Omron CX-Programmer project RECYCLING_EPP (CX-Programmer 9.81)

# PLC NewPLC1: CP1L-E EL

## Global symbols (name address type ; comment)
D101 CHANNEL  ; Valore proporzionale da 0001 a 270F
D102 CHANNEL  ; Valore Integrale da 0001 a 1FFF
D500 CHANNEL  ; Configurazione MAD Analogica
H10.01 BOOL  ; PID error
T0000 BOOL  ; TON Sensore Livello
T0001 BOOL  ; TOF Sensore livello
T0002 BOOL  ; K1 TON
T0003 BOOL  ; K1 TOF
T0004 BOOL  ; KM2 TON
T0005 BOOL  ; KM2 TOF
T0006 BOOL  ; KM3 TON
T0007 BOOL  ; KM3 TOF
W0 CHANNEL  ; Word Allarmi
Out_K1_Bis 100.00 BOOL

## Program NuovoProgramma1 (cyclic task 0)
; Conversione e controllo valori immessi dal touch screen
Local symbols
Allarme W2.00 BOOL  ; PLC in allarme
Errore_Fungo W0.06 BOOL  ; Fungo emergenza premuto
Errore_Inverter W0.10 BOOL  ; Inverter in allarme
Errore_K1_non_apre W0.00 BOOL  ; K1 non viene diseccitato
Errore_K1_non_chiude W0.01 BOOL  ; K1 non viene eccitato
Errore_KM2_non_apre W0.02 BOOL  ; KM2 non viene diseccitato
Errore_KM2_non_chiude W0.03 BOOL  ; KM2 non viene eccitato
Errore_KM3_non_apre W0.04 BOOL  ; KM3 non viene diseccitato
Errore_KM3_non_chiude W0.05 BOOL  ; KM3 non viene eccitato
Errore_QM1 W0.07 BOOL  ; Magnetotermico QM1
Errore_QM2 W0.08 BOOL  ; Magnetotermico QM2
Errore_QM3 W0.09 BOOL  ; Magnetotermico QM3
Inp_Errore_Inverter 0.09 BOOL  ; Inverter in errore
Inp_Fungo 0.00 BOOL  ; Fungo di emergenza
Inp_K1_24OUT 0.10 BOOL  ; Ho la 24OUT in ingresso
Inp_KM2 0.07 BOOL  ; Input KM2
Inp_KM3 0.08 BOOL  ; Input KM3
Inp_QM1 0.04 BOOL  ; Input QM1
Inp_QM2 0.05 BOOL  ; Input QM2
Inp_QM3 0.06 BOOL  ; Input QM3
Inp_Sensore_Livello 0.03 BOOL  ; Fotocellula presenza materiale
Inp_Start 0.01 BOOL  ; Pulsante Start
Inp_Stop 0.02 BOOL  ; Pulsante Stop
Livello_Materiale_Pieno W2.01 BOOL  ; Sensore livello con TON e TOF
Out_Frequenza_Inverter 101 UINT  ; Frequenza a cui far girare l'inverter
Out_Inverter 100.03 BOOL  ; Attivazione inverter
Out_K1 100.00 BOOL  ; Attivazione marcia
Out_K1_Bis 100.02 BOOL  ; Attivazione marcia
Out_KM2 100.04 BOOL  ; Attivazione KM2
Out_KM3 100.05 BOOL  ; Attivazione KM3
Out_Reset_Inverter 100.01 BOOL  ; Resetto l'errore dell'Inverter
Par_Percentuale W1 UINT  ; Percentuale di riciclato (da 0 a 50%)
Par_Percentuale_Rem D1000 UINT  ; Percentuale di riciclato (da 0 a 50%) in memoria remanent
Reset_Allarmi W2.02 BOOL  ; Richiesta da pannello di reset degli allarmi

### Section Controllo_Parametri

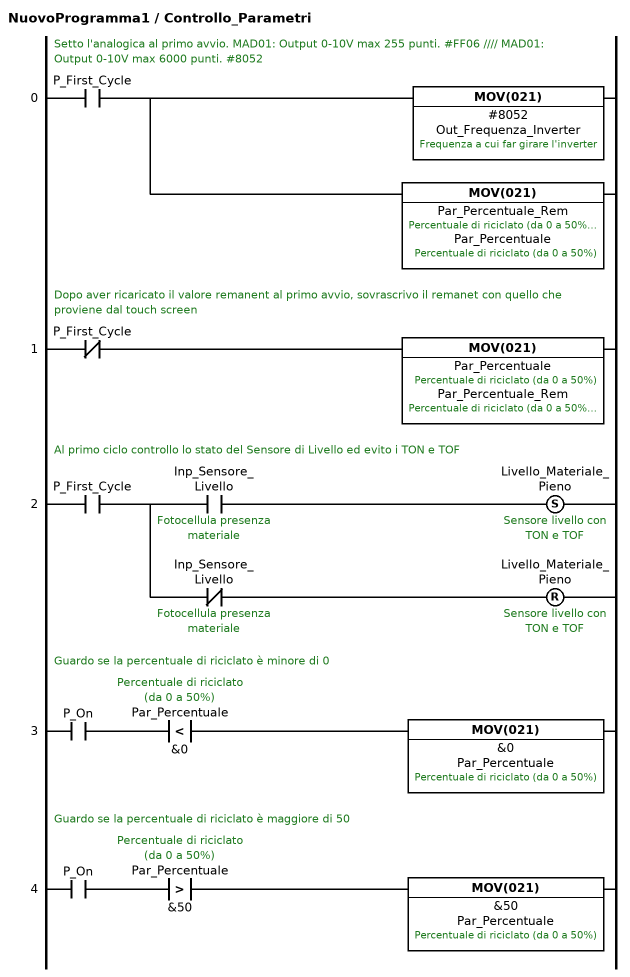
; rung 0: Setto l'analogica al primo avvio. MAD01: Output 0-10V max 255 punti. #FF06 //// MAD01: Output 0-10V max 6000 punti. #8052
LD P_First_Cycle
MOV(021) #8052 Out_Frequenza_Inverter  ; Frequenza a cui far girare l'inverter
MOV(021) Par_Percentuale_Rem Par_Percentuale  ; Percentuale di riciclato (da 0 a 50%) in memoria remanent, Percentuale di riciclato (da 0 a 50%)
; rung 1: Dopo aver ricaricato il valore remanent al primo avvio, sovrascrivo il remanet con quello che proviene dal touch screen
LDNOT P_First_Cycle
MOV(021) Par_Percentuale Par_Percentuale_Rem  ; Percentuale di riciclato (da 0 a 50%), Percentuale di riciclato (da 0 a 50%) in memoria remanent
; rung 2: Al primo ciclo controllo lo stato del Sensore di Livello ed evito i TON e TOF
LD P_First_Cycle
OUT TR0
AND Inp_Sensore_Livello  ; Fotocellula presenza materiale
SET Livello_Materiale_Pieno  ; Sensore livello con TON e TOF
LD TR0
ANDNOT Inp_Sensore_Livello  ; Fotocellula presenza materiale
RSET Livello_Materiale_Pieno  ; Sensore livello con TON e TOF
; rung 3: Guardo se la percentuale di riciclato è minore di 0
LD P_On
AND<(310) Par_Percentuale &0  ; Percentuale di riciclato (da 0 a 50%)
MOV(021) &0 Par_Percentuale  ; Percentuale di riciclato (da 0 a 50%)
; rung 4: Guardo se la percentuale di riciclato è maggiore di 50
LD P_On
AND>(320) Par_Percentuale &50  ; Percentuale di riciclato (da 0 a 50%)
MOV(021) &50 Par_Percentuale  ; Percentuale di riciclato (da 0 a 50%)

### Section Logica

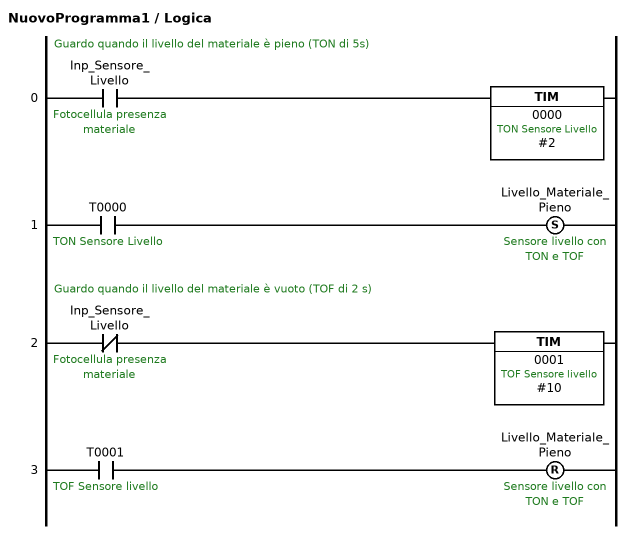
; rung 0: Guardo quando il livello del materiale è pieno (TON di 5s)
LD Inp_Sensore_Livello  ; Fotocellula presenza materiale
TIM 0000 #2  ; TON Sensore Livello
; rung 1
LD T0000  ; TON Sensore Livello
SET Livello_Materiale_Pieno  ; Sensore livello con TON e TOF
; rung 2: Guardo quando il livello del materiale è vuoto (TOF di 2 s)
LDNOT Inp_Sensore_Livello  ; Fotocellula presenza materiale
TIM 0001 #10  ; TOF Sensore livello
; rung 3
LD T0001  ; TOF Sensore livello
RSET Livello_Materiale_Pieno  ; Sensore livello con TON e TOF

### Section Diagnostica

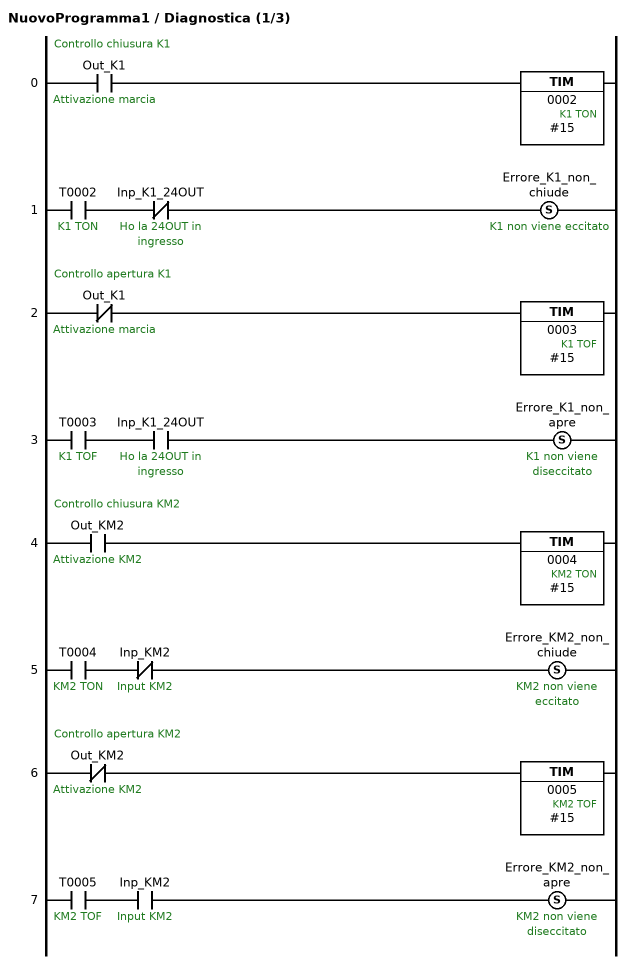
; rung 0: Controllo chiusura K1
LD Out_K1  ; Attivazione marcia
TIM 0002 #15  ; K1 TON
; rung 1
LD T0002  ; K1 TON
ANDNOT Inp_K1_24OUT  ; Ho la 24OUT in ingresso
SET Errore_K1_non_chiude  ; K1 non viene eccitato
; rung 2: Controllo apertura K1
LDNOT Out_K1  ; Attivazione marcia
TIM 0003 #15  ; K1 TOF
; rung 3
LD T0003  ; K1 TOF
AND Inp_K1_24OUT  ; Ho la 24OUT in ingresso
SET Errore_K1_non_apre  ; K1 non viene diseccitato
; rung 4: Controllo chiusura KM2
LD Out_KM2  ; Attivazione KM2
TIM 0004 #15  ; KM2 TON
; rung 5
LD T0004  ; KM2 TON
ANDNOT Inp_KM2  ; Input KM2
SET Errore_KM2_non_chiude  ; KM2 non viene eccitato
; rung 6: Controllo apertura KM2
LDNOT Out_KM2  ; Attivazione KM2
TIM 0005 #15  ; KM2 TOF
; rung 7
LD T0005  ; KM2 TOF
AND Inp_KM2  ; Input KM2
SET Errore_KM2_non_apre  ; KM2 non viene diseccitato

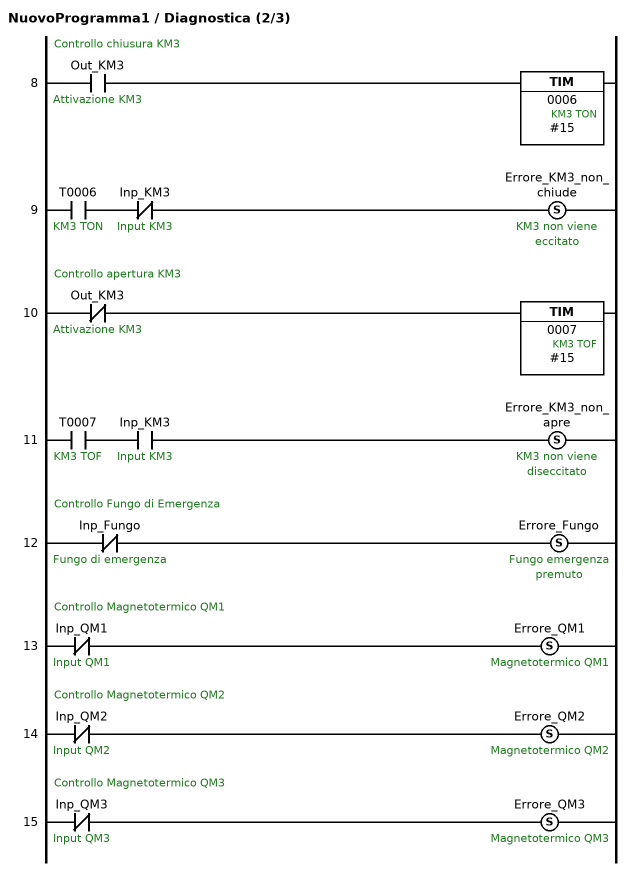
; rung 8: Controllo chiusura KM3
LD Out_KM3  ; Attivazione KM3
TIM 0006 #15  ; KM3 TON
; rung 9
LD T0006  ; KM3 TON
ANDNOT Inp_KM3  ; Input KM3
SET Errore_KM3_non_chiude  ; KM3 non viene eccitato
; rung 10: Controllo apertura KM3
LDNOT Out_KM3  ; Attivazione KM3
TIM 0007 #15  ; KM3 TOF
; rung 11
LD T0007  ; KM3 TOF
AND Inp_KM3  ; Input KM3
SET Errore_KM3_non_apre  ; KM3 non viene diseccitato
; rung 12: Controllo Fungo di Emergenza
LDNOT Inp_Fungo  ; Fungo di emergenza
SET Errore_Fungo  ; Fungo emergenza premuto
; rung 13: Controllo Magnetotermico QM1
LDNOT Inp_QM1  ; Input QM1
SET Errore_QM1  ; Magnetotermico QM1
; rung 14: Controllo Magnetotermico QM2
LDNOT Inp_QM2  ; Input QM2
SET Errore_QM2  ; Magnetotermico QM2
; rung 15: Controllo Magnetotermico QM3
LDNOT Inp_QM3  ; Input QM3
SET Errore_QM3  ; Magnetotermico QM3

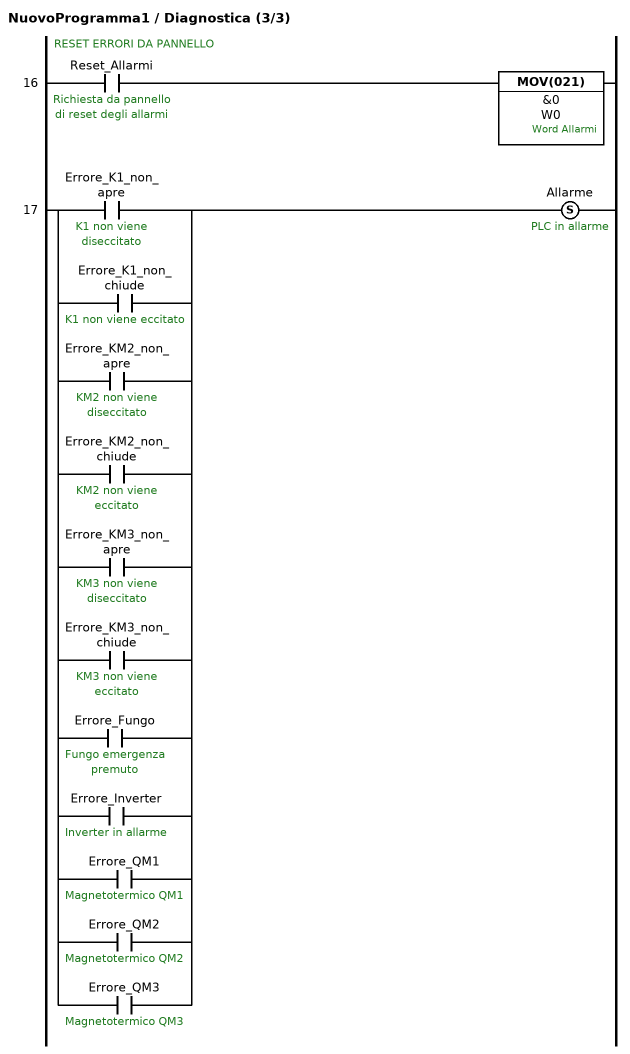
; rung 16: RESET ERRORI DA PANNELLO
LD Reset_Allarmi  ; Richiesta da pannello di reset degli allarmi
MOV(021) &0 W0  ; Word Allarmi
; rung 17
LD Errore_K1_non_apre  ; K1 non viene diseccitato
OR Errore_K1_non_chiude  ; K1 non viene eccitato
OR Errore_KM2_non_apre  ; KM2 non viene diseccitato
OR Errore_KM2_non_chiude  ; KM2 non viene eccitato
OR Errore_KM3_non_apre  ; KM3 non viene diseccitato
OR Errore_KM3_non_chiude  ; KM3 non viene eccitato
OR Errore_Fungo  ; Fungo emergenza premuto
OR Errore_Inverter  ; Inverter in allarme
OR Errore_QM1  ; Magnetotermico QM1
OR Errore_QM2  ; Magnetotermico QM2
OR Errore_QM3  ; Magnetotermico QM3
SET Allarme  ; PLC in allarme

### Section I_O

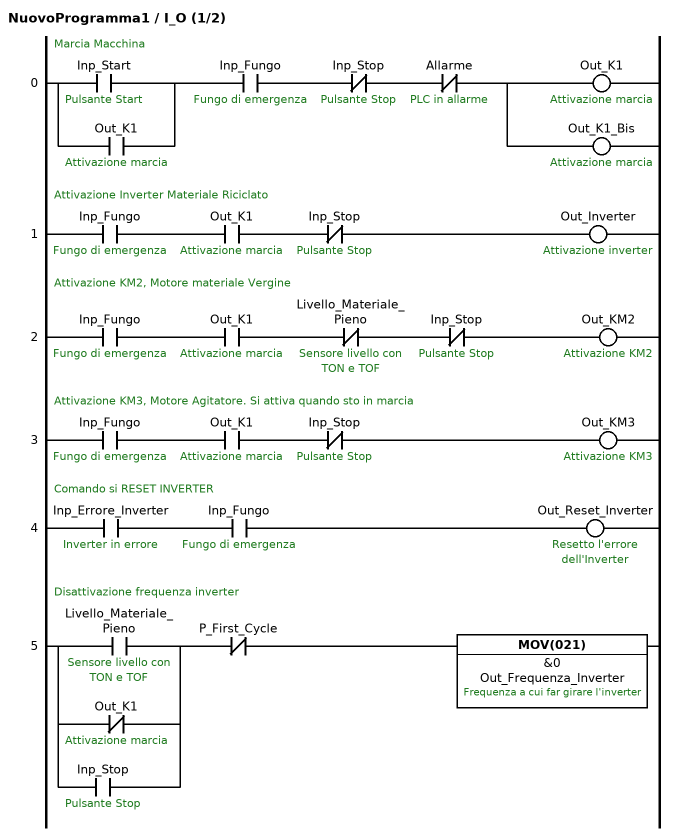
; rung 0: Marcia Macchina
LD Inp_Start  ; Pulsante Start
OR Out_K1  ; Attivazione marcia
AND Inp_Fungo  ; Fungo di emergenza
ANDNOT Inp_Stop  ; Pulsante Stop
ANDNOT Allarme  ; PLC in allarme
OUT Out_K1  ; Attivazione marcia
OUT Out_K1_Bis  ; Attivazione marcia
; rung 1: Attivazione Inverter Materiale Riciclato
LD Inp_Fungo  ; Fungo di emergenza
AND Out_K1  ; Attivazione marcia
ANDNOT Inp_Stop  ; Pulsante Stop
OUT Out_Inverter  ; Attivazione inverter
; rung 2: Attivazione KM2, Motore materiale Vergine
LD Inp_Fungo  ; Fungo di emergenza
AND Out_K1  ; Attivazione marcia
ANDNOT Livello_Materiale_Pieno  ; Sensore livello con TON e TOF
ANDNOT Inp_Stop  ; Pulsante Stop
OUT Out_KM2  ; Attivazione KM2
; rung 3: Attivazione KM3, Motore Agitatore. Si attiva quando sto in marcia
LD Inp_Fungo  ; Fungo di emergenza
AND Out_K1  ; Attivazione marcia
ANDNOT Inp_Stop  ; Pulsante Stop
OUT Out_KM3  ; Attivazione KM3
; rung 4: Comando si RESET INVERTER
LD Inp_Errore_Inverter  ; Inverter in errore
AND Inp_Fungo  ; Fungo di emergenza
OUT Out_Reset_Inverter  ; Resetto l'errore dell'Inverter
; rung 5: Disattivazione frequenza inverter
LD Livello_Materiale_Pieno  ; Sensore livello con TON e TOF
ORNOT Out_K1  ; Attivazione marcia
OR Inp_Stop  ; Pulsante Stop
ANDNOT P_First_Cycle
MOV(021) &0 Out_Frequenza_Inverter  ; Frequenza a cui far girare l'inverter

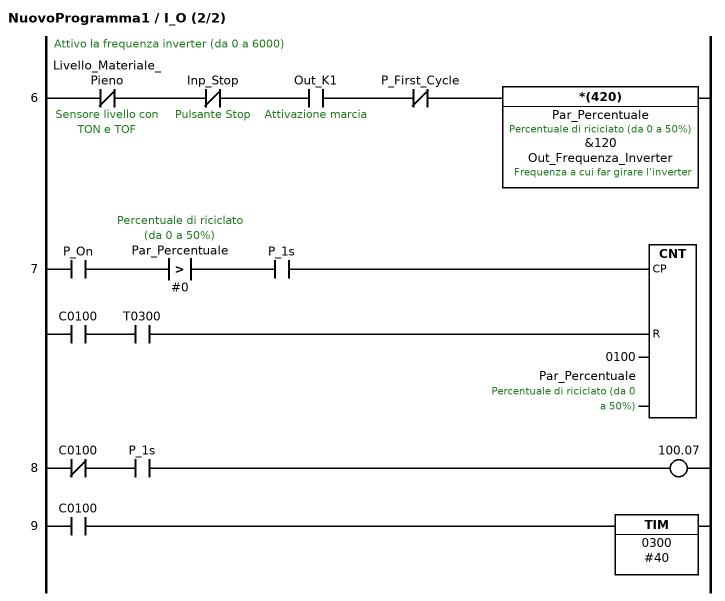
; rung 6: Attivo la frequenza inverter (da 0 a 6000)
LDNOT Livello_Materiale_Pieno  ; Sensore livello con TON e TOF
ANDNOT Inp_Stop  ; Pulsante Stop
AND Out_K1  ; Attivazione marcia
ANDNOT P_First_Cycle
*(420) Par_Percentuale &120 Out_Frequenza_Inverter  ; Percentuale di riciclato (da 0 a 50%), Frequenza a cui far girare l'inverter
; rung 7
LD P_On
AND>(320) Par_Percentuale #0  ; Percentuale di riciclato (da 0 a 50%)
AND P_1s
LD C0100
AND T0300
CNT 0100 Par_Percentuale  ; Percentuale di riciclato (da 0 a 50%)
; rung 8
LDNOT C0100
AND P_1s
OUT 100.07
; rung 9
LD C0100
TIM 0300 #40

### Section END
; rung 0
END(001)